# B&R Automation Studio project Template (part 2)

#### slave.fun - functions
```iecst
(********************************************************************
 * COPYRIGHT -- Bernecker + Rainer
 ********************************************************************
 * Program: Slave_00
 * File: Slave_00.fun
 * Author: reischlj
 * Created: March 09, 2011
 ********************************************************************
 * Functions and function blocks of program Slave_00
 ********************************************************************)

FUNCTION Labeler : BOOL
	VAR_INPUT
		Axis : UDINT;
	END_VAR
	VAR_IN_OUT
		AutData : MC_AUTDATA_TYP;
	END_VAR
END_FUNCTION

FUNCTION CrossCutter : BOOL
	VAR_INPUT
		Axis : UDINT;
	END_VAR
	VAR_IN_OUT
		AutData : MC_AUTDATA_TYP;
	END_VAR
END_FUNCTION

FUNCTION FlyingSaw : BOOL
	VAR_INPUT
		Axis  : UDINT;
	END_VAR
	VAR_IN_OUT
		AutData : MC_AUTDATA_TYP;
	END_VAR
END_FUNCTION
```

#### Labeler.st - function
```iecst
(********************************************************************
 * COPYRIGHT -- Bernecker + Rainer
 ********************************************************************
 * PROGRAM: Slave
 * File: Labeler.st
 * Author: Bernecker + Rainer
 * Created: March 01, 2011
 *******************************************************************)

FUNCTION Labeler
    (*general automat parameter*)
        AutData.Master              := Axis;

        AutData.MaxMasterVelocity   := 1000;

    (*Automat STATE 0 Basis State*)

        AutData.State[0].Event[0].Type      := ncST_END;

        AutData.State[0].Event[0].Attribute := ncAT_ONCE;

        AutData.State[0].Event[0].NextState := 1;

    (*Automat STATE 1 Standstill*)

        AutData.State[1].CamProfileIndex    := 16#FFFF;

        AutData.State[1].MasterFactor       := 200;

        AutData.State[1].SlaveFactor        := 0;

        AutData.State[1].CompMode           := ncONLYCOMP;

        AutData.State[1].MasterCompDistance := 800;

        AutData.State[1].SlaveCompDistance  := 0;

        AutData.State[1].Event[0].Type      := ncTRIGGER1+ncP_EDGE;

        AutData.State[1].Event[0].Attribute := ncST_END;

        AutData.State[1].Event[0].NextState := 2;

        AutData.State[1].Event[1].Type      := ncST_END;

        AutData.State[1].Event[1].Attribute := ncST_END;

        AutData.State[1].Event[1].NextState := 1;

    (*Automat STATE 2 Labeling with half compensation*)

        AutData.State[2].CamProfileIndex    := 16#FFFF;

        AutData.State[2].MasterFactor       := 200;

        AutData.State[2].SlaveFactor        := 200;

        AutData.State[2].CompMode           := ncONLYCOMP;
        AutData.State[2].MasterCompDistance := 800;

        AutData.State[2].SlaveCompDistance  := 400;

        AutData.State[2].Event[0].Type      := ncTRIGGER1+ncP_EDGE;

        AutData.State[2].Event[0].Attribute := ncST_END;

        AutData.State[2].Event[0].NextState := 3;

        AutData.State[2].Event[1].Type      := ncST_END;

        AutData.State[2].Event[1].Attribute := ncST_END;

        AutData.State[2].Event[1].NextState := 4;

    (*Automat STATE 3 Labeling *)

        AutData.State[3].CamProfileIndex    := 16#FFFF;

        AutData.State[3].MasterFactor       := 200;

        AutData.State[3].SlaveFactor        := 200;

        AutData.State[3].CompMode           := ncONLYCOMP;

        AutData.State[3].MasterCompDistance := 800;

        AutData.State[3].SlaveCompDistance  := 800;

        AutData.State[3].Event[0].Type      := ncTRIGGER1+ncP_EDGE;

        AutData.State[3].Event[0].Attribute := ncST_END;

        AutData.State[3].Event[0].NextState := 3;

        AutData.State[3].Event[1].Type      := ncST_END;
		AutData.State[3].Event[1].Attribute := ncST_END;
		AutData.State[3].Event[1].NextState := 4;

    (*Automat STATE 4 Return to starting position*)
        AutData.State[4].CamProfileIndex    := 16#FFFF;
        AutData.State[4].MasterFactor       := 200;
        AutData.State[4].SlaveFactor        := 0;
        AutData.State[4].CompMode           := ncONLYCOMP;
        AutData.State[4].MasterCompDistance := 800;
        AutData.State[4].SlaveCompDistance  := 400;

        AutData.State[4].Event[0].Type      := ncTRIGGER1+ncP_EDGE;
        AutData.State[4].Event[0].Attribute := ncST_END;
        AutData.State[4].Event[0].NextState := 2;

        AutData.State[4].Event[1].Type      := ncST_END;
        AutData.State[4].Event[1].Attribute := ncST_END;
        AutData.State[4].Event[1].NextState := 1;

        Labeler := TRUE;
END_FUNCTION
```

#### CrossCutter.st - function
```iecst
(********************************************************************
 * COPYRIGHT -- Bernecker + Rainer
 ********************************************************************
 * PROGRAM: Slave
 * File: CrossCutter.st
 * Author: Bernecker + Rainer
 * Created: March 01, 2011
 *******************************************************************)

FUNCTION CrossCutter
    (*general automat parameter*)
        AutData.Master              := Axis;

        AutData.MaxMasterVelocity   := 1000;

    (*Automat STATE 0 Basis State*)

        AutData.State[0].Event[0].Type      := ncST_END;

        AutData.State[0].Event[0].Attribute := ncAT_ONCE;

        AutData.State[0].Event[0].NextState := 1;

    (*Automat STATE 1 Standstill*)

        AutData.State[1].CamProfileIndex    := 16#FFFE;

        AutData.State[1].MasterFactor       := 200;

        AutData.State[1].SlaveFactor        := 0;
        AutData.State[1].CompMode           := ncWITH_CAM;
        AutData.State[1].MasterCompDistance := 1000;
        AutData.State[1].SlaveCompDistance  := 0;

        AutData.State[1].Event[0].Type      := ncSIGNAL1;
        AutData.State[1].Event[0].Attribute := ncAT_ONCE;
        AutData.State[1].Event[0].NextState := 2;

    (*Automat STATE 2 Move Slave to Cutting Position*)
        AutData.State[2].CamProfileIndex    := 16#FFFF;
        AutData.State[2].MasterFactor       := 200;
        AutData.State[2].SlaveFactor        := 200;
        AutData.State[2].CompMode           := ncWITH_CAM;
        AutData.State[2].MasterCompDistance := 500;
        AutData.State[2].SlaveCompDistance  := 1800;

        AutData.State[2].Event[0].Type      := ncST_END;
        AutData.State[2].Event[0].Attribute := ncST_END;
        AutData.State[2].Event[0].NextState := 3;

    (*Automat STATE 3 Execute one cut every master period*)
        AutData.State[3].CamProfileIndex    := 16#FFFF;
        AutData.State[3].MasterFactor       := 200;
        AutData.State[3].SlaveFactor        := 200;
        AutData.State[3].CompMode           := ncWITH_CAM;
        AutData.State[3].MasterCompDistance := 1000;
        AutData.State[3].SlaveCompDistance  := 3600;

        AutData.State[3].Event[0].Type      := ncSIGNAL2;
        AutData.State[3].Event[0].Attribute := ncST_END;
        AutData.State[3].Event[0].NextState := 4;

        AutData.State[3].Event[1].Type      := ncST_END;
        AutData.State[3].Event[1].Attribute := ncST_END;
        AutData.State[3].Event[1].NextState := 3;

    (*Automat STATE 4 Stop Motion at Starting Point*)
        AutData.State[4].CamProfileIndex    := 16#FFFF;
        AutData.State[4].MasterFactor       := 200;
        AutData.State[4].SlaveFactor        := 0;
        AutData.State[4].CompMode           := ncWITH_CAM;
        AutData.State[4].MasterCompDistance := 500;
        AutData.State[4].SlaveCompDistance  := 1800;

        AutData.State[4].Event[0].Type      := ncST_END;
        AutData.State[4].Event[0].Attribute := ncST_END;
        AutData.State[4].Event[0].NextState := 1;

        CrossCutter := TRUE;
END_FUNCTION
```

#### FlyingSaw.st - function
```iecst
(********************************************************************
 * COPYRIGHT -- Bernecker + Rainer
 ********************************************************************
 * PROGRAM: Slave
 * File: FlyingSaw.st
 * Author: Bernecker + Rainer
 * Created: March 01, 2011
 *******************************************************************)

FUNCTION FlyingSaw
    (*general automat parameters*)
        AutData.Master              := Axis;

        AutData.StartPosition       := 0;

        AutData.StartInterval       := 1000;

        AutData.MaxMasterVelocity   := 1000;

    (*Automat STATE 0 Basis State*)

        AutData.State[0].Event[0].Type      := ncST_END;

        AutData.State[0].Event[0].Attribute := ncAT_ONCE;

        AutData.State[0].Event[0].NextState := 1;

    (*Automat STATE 1 Standstill*)

        AutData.State[1].CamProfileIndex    := 16#FFFF;

        AutData.State[1].MasterFactor       := 200;

        AutData.State[1].SlaveFactor        := 0;

        AutData.State[1].CompMode           := ncONLYCOMP;

        AutData.State[1].MasterCompDistance := 800;

        AutData.State[1].SlaveCompDistance  := 0;

        AutData.State[1].Event[0].Type      := ncS_START;

        AutData.State[1].Event[0].Attribute := ncAT_ONCE;

        AutData.State[1].Event[0].NextState := 2;

    (*Autoamt STATE 2 Synchronous movement*)
        AutData.State[2].CamProfileIndex    := 16#FFFF;
        AutData.State[2].MasterFactor       := 500;
        AutData.State[2].SlaveFactor        := 500;
        AutData.State[2].CompMode           := ncONLYCOMP;
        AutData.State[2].MasterCompDistance := 100;
        AutData.State[2].SlaveCompDistance  := 100;

        AutData.State[2].Event[0].Type      := ncST_END;
        AutData.State[2].Event[0].Attribute := ncST_END;
        AutData.State[2].Event[0].NextState := 3;

    (*Automat STATE 3 Return to starting position*)
        AutData.State[3].CamProfileIndex    := 16#FFFF;
        AutData.State[3].MasterFactor       := 100;
        AutData.State[3].SlaveFactor        := 0;
        AutData.State[3].CompMode           := ncONLYCOMP;
        AutData.State[3].MasterCompDistance := 800;
        AutData.State[3].SlaveCompDistance  := -600;

        AutData.State[3].Event[0].Type      := ncST_END;
        AutData.State[3].Event[0].Attribute := ncST_END;
        AutData.State[3].Event[0].NextState := 1;

        FlyingSaw := TRUE;
END_FUNCTION
```

### Program Logical/LibACP10MC_MotionControl_ST/ErrorHandling (IEC) - error handling task

#### errorHandlingCyclic.st - Cyclic code
```iecst
(********************************************************************
 * COPYRIGHT -- Bernecker + Rainer
 ********************************************************************
 * Program: ErrorHandling
 * File: errorHandlingCyclic.st
 * Author: Bernecker + Rainer
 * Created: March 01, 2011
 ********************************************************************
 * Implementation of program Errorhandling
 ********************************************************************)

PROGRAM _CYCLIC

(******************************ERROR_CHECK***************************)
(* check if one of the used FBs reports an error *)
IF ((MC_BR_AxisErrorCollector_0.Error = TRUE) OR (MC_Reset_0.Error = TRUE)) THEN
    ErrorStep := STATE_INTERNAL_ERROR;
END_IF

FOR configAxisIndex := 0 TO TOTAL_AXES BY 1 DO
    IF ((MC_BR_ReadAxisError_0[configAxisIndex].Error = TRUE) OR (MC_ReadStatus_0[configAxisIndex].Error = TRUE)) THEN
        ErrorStep := STATE_INTERNAL_ERROR;
        EXIT;
    END_IF
END_FOR

CASE ErrorStep OF

(**************************** CONFIGURATE_FBS ***********************)
    STATE_CONFIG_FBS: (* configurate the used FBs for the error handling *)
        MC_BR_AxisErrorCollector_0.Axis := mcALL_AXES;
        MC_BR_AxisErrorCollector_0.Enable := TRUE;

        (* configuration the MC_BR_ReadAxisError_0-FBs for all single axes *)
        FOR axisIndex := 0 TO (AXIS_MAX_INDEX) BY 1 DO
            MC_BR_ReadAxisError_0[axisIndex].Axis := AxisRef[axisIndex];
            MC_BR_ReadAxisError_0[axisIndex].Enable := TRUE;
            MC_BR_ReadAxisError_0[axisIndex].Configuration.Format := mcWRAP;
            MC_BR_ReadAxisError_0[axisIndex].Configuration.LineLength := SIZEOF(Axis[axisIndex].Error.ErrorText[0]);
            MC_BR_ReadAxisError_0[axisIndex].Configuration.DataLength := SIZEOF(Axis[axisIndex].Error.ErrorText);
            MC_BR_ReadAxisError_0[axisIndex].Configuration.DataAddress := ADR(Axis[axisIndex].Error.ErrorText[0]);
            MC_BR_ReadAxisError_0[axisIndex].Configuration.DataObjectName :='acp10etxen';
            MC_BR_ReadAxisError_0[axisIndex].Mode := mcTEXT;

            MC_ReadStatus_0[axisIndex].Axis := AxisRef[axisIndex];
            MC_ReadStatus_0[axisIndex].Enable := TRUE;
        END_FOR

        (* configuration the MC_BR_ReadAxisError_0-FBs for all master axes *)
        FOR masterIndex := 0 TO (MASTER_MAX_INDEX) BY 1 DO
            MC_BR_ReadAxisError_0[masterIndex+AXIS_NUMBER].Axis := MasterRef[masterIndex];
            MC_BR_ReadAxisError_0[masterIndex+AXIS_NUMBER].Enable := TRUE;
            MC_BR_ReadAxisError_0[masterIndex+AXIS_NUMBER].Configuration.Format := mcWRAP;
            MC_BR_ReadAxisError_0[masterIndex+AXIS_NUMBER].Configuration.LineLength := SIZEOF(Master[masterIndex].Error.ErrorText[0]);
            MC_BR_ReadAxisError_0[masterIndex+AXIS_NUMBER].Configuration.DataLength := SIZEOF(Master[masterIndex].Error.ErrorText);
            MC_BR_ReadAxisError_0[masterIndex+AXIS_NUMBER].Configuration.DataAddress := ADR(Master[masterIndex].Error.ErrorText[0]);
            MC_BR_ReadAxisError_0[masterIndex+AXIS_NUMBER].Configuration.DataObjectName := 'acp10etxen';
            MC_BR_ReadAxisError_0[masterIndex+AXIS_NUMBER].Mode := mcTEXT;

            MC_ReadStatus_0[masterIndex+AXIS_NUMBER].Axis := MasterRef[masterIndex];
            MC_ReadStatus_0[masterIndex+AXIS_NUMBER].Enable := TRUE;
        END_FOR

        (* configuration the MC_BR_ReadAxisError_0-FBs for all slave axes *)
        FOR slaveIndex := 0 TO (SLAVE_MAX_INDEX) BY 1 DO
            MC_BR_ReadAxisError_0[slaveIndex+AXIS_NUMBER+MASTER_NUMBER].Axis := SlaveRef[slaveIndex];
            MC_BR_ReadAxisError_0[slaveIndex+AXIS_NUMBER+MASTER_NUMBER].Enable := TRUE;
            MC_BR_ReadAxisError_0[slaveIndex+AXIS_NUMBER+MASTER_NUMBER].Configuration.Format := mcWRAP;
            MC_BR_ReadAxisError_0[slaveIndex+AXIS_NUMBER+MASTER_NUMBER].Configuration.LineLength := SIZEOF(Slave[slaveIndex].Error.ErrorText[0]);
            MC_BR_ReadAxisError_0[slaveIndex+AXIS_NUMBER+MASTER_NUMBER].Configuration.DataLength := SIZEOF(Slave[slaveIndex].Error.ErrorText);
            MC_BR_ReadAxisError_0[slaveIndex+AXIS_NUMBER+MASTER_NUMBER].Configuration.DataAddress := ADR(Slave[slaveIndex].Error.ErrorText[0]);
            MC_BR_ReadAxisError_0[slaveIndex+AXIS_NUMBER+MASTER_NUMBER].Configuration.DataObjectName := 'acp10etxen';
            MC_BR_ReadAxisError_0[slaveIndex+AXIS_NUMBER+MASTER_NUMBER].Mode := mcTEXT;

            MC_ReadStatus_0[slaveIndex+AXIS_NUMBER+MASTER_NUMBER].Axis := SlaveRef[slaveIndex];
            MC_ReadStatus_0[slaveIndex+AXIS_NUMBER+MASTER_NUMBER].Enable := TRUE;
        END_FOR

        (* configuration the MC_BR_ReadAxisError_0-FBs for all power supply module *)
        FOR psmIndex := 0 TO (PSM_MAX_INDEX) BY 1 DO
            MC_BR_ReadAxisError_0[psmIndex+AXIS_NUMBER+MASTER_NUMBER+SLAVE_NUMBER].Axis := PsmRef[psmIndex];
            MC_BR_ReadAxisError_0[psmIndex+AXIS_NUMBER+MASTER_NUMBER+SLAVE_NUMBER].Enable := TRUE;
            MC_BR_ReadAxisError_0[psmIndex+AXIS_NUMBER+MASTER_NUMBER+SLAVE_NUMBER].Configuration.Format := mcWRAP;
            MC_BR_ReadAxisError_0[psmIndex+AXIS_NUMBER+MASTER_NUMBER+SLAVE_NUMBER].Configuration.LineLength := SIZEOF(PowerSupply[psmIndex].Error.ErrorText[0]);
            MC_BR_ReadAxisError_0[psmIndex+AXIS_NUMBER+MASTER_NUMBER+SLAVE_NUMBER].Configuration.DataLength := SIZEOF(PowerSupply[psmIndex].Error.ErrorText);
            MC_BR_ReadAxisError_0[psmIndex+AXIS_NUMBER+MASTER_NUMBER+SLAVE_NUMBER].Configuration.DataAddress := ADR(PowerSupply[psmIndex].Error.ErrorText[0]);
            MC_BR_ReadAxisError_0[psmIndex+AXIS_NUMBER+MASTER_NUMBER+SLAVE_NUMBER].Configuration.DataObjectName := 'acp10etxen';
            MC_BR_ReadAxisError_0[psmIndex+AXIS_NUMBER+MASTER_NUMBER+SLAVE_NUMBER].Mode := mcTEXT;

            MC_ReadStatus_0[psmIndex+AXIS_NUMBER+MASTER_NUMBER+SLAVE_NUMBER].Axis := PsmRef[psmIndex];
            MC_ReadStatus_0[psmIndex+AXIS_NUMBER+MASTER_NUMBER+SLAVE_NUMBER].Enable := TRUE;
        END_FOR

        ErrorStep := STATE_WAIT;
        AcknowledgeStep := STATE_ERROR_SCAN;

        (* End of STATE_CONFIG_FBS *)

(*************************** CHECK_AXES_FOR_ERROR *******************)
    STATE_WAIT: (* check if at least on one of the axes an error occured *)
        IF ((MC_BR_AxisErrorCollector_0.AxisError = TRUE) OR
            (MC_BR_AxisErrorCollector_0.AxisWarning = TRUE) OR
            (MC_BR_AxisErrorCollector_0.FunctionBlockError = TRUE) OR
            (MC_BR_AxisErrorCollector_0.Errorstop = TRUE)) THEN
              ErrorStep := STATE_ERROR_HANDLING;
        ELSE
            GlobalError.AxisTyp := '';
            GlobalError.AxisIndex := 0;
            GlobalError.ErrorRecord.Info := 0;
            GlobalError.ErrorRecord.Number := 0;
            GlobalError.ErrorRecord.ParID := 0;
            GlobalError.ErrorText[0] := '';
            GlobalError.ErrorText[1] := '';
            GlobalError.ErrorText[2] := '';
            GlobalError.ErrorText[3] := '';
        END_IF

        (* End of STATE_WAIT *)

(**************************** HANDLE_ACTIVE_ERRORS ******************)
    STATE_ERROR_HANDLING: (* check witch axis is in ErrorStop and withc axes has to be stopped *)
        (* check if a single axis has to be stopped *)
        FOR axisIndex := 0 TO (AXIS_MAX_INDEX) BY 1 DO
            IF (MC_ReadStatus_0[axisIndex].Errorstop = TRUE) THEN
                Axis[axisIndex].Command.Stop := TRUE;
            END_IF
        END_FOR

        (* check if the master slave combination has to be stopped *)
        FOR masterIndex := 0 TO (MASTER_MAX_INDEX) BY 1 DO
            IF (MC_ReadStatus_0[masterIndex+AXIS_NUMBER].Errorstop = TRUE) THEN
                FOR masterIndex := 0 TO (MASTER_MAX_INDEX) BY 1 DO
                    Master[masterIndex].Command.Stop := TRUE;
                END_FOR

                FOR slaveIndex := 0 TO (SLAVE_MAX_INDEX) BY 1 DO
                    Slave[slaveIndex].Command.Stop := TRUE;
                END_FOR
            END_IF
        END_FOR

        (* check if the master slave combination has to be stopped *)
        FOR slaveIndex := 0 TO (SLAVE_MAX_INDEX) BY 1 DO
            IF  (MC_ReadStatus_0[slaveIndex+AXIS_NUMBER+MASTER_NUMBER].Errorstop = TRUE) THEN
                FOR masterIndex := 0 TO (MASTER_MAX_INDEX) BY 1 DO
                    Master[masterIndex].Command.Stop := TRUE;
                END_FOR

                FOR slaveIndex := 0 TO (SLAVE_MAX_INDEX) BY 1 DO
                    Slave[slaveIndex].Command.Stop := TRUE;
                END_FOR
            END_IF
        END_FOR

    (******************* STEP_SEQUENCE OF ERROR ACKNOWLEDGE *************)
    CASE AcknowledgeStep OF
        (************************** SEARCH FOR ERRORS ***********************)
        STATE_ERROR_SCAN: (* check if an error is active on one of the axis *)
            ErrorStep := STATE_WAIT;
            FOR totalAxisIndex := 0 TO (TOTAL_AXES-1) BY 1 DO
                IF ((MC_BR_ReadAxisError_0[totalAxisIndex].AxisErrorCount > 0) OR
                    (MC_BR_ReadAxisError_0[totalAxisIndex].AxisWarningCount > 0) OR
                    (MC_BR_ReadAxisError_0[totalAxisIndex].FunctionBlockErrorCount > 0)) THEN
                    AcknowledgeStep := STATE_ERROR_ACKNOWLEDGE;
                    ErrorStep := STATE_ERROR_HANDLING;
                    EXIT;
                ELSIF (MC_ReadStatus_0[totalAxisIndex].Errorstop = TRUE) THEN
                    AcknowledgeStep := STATE_RESET;
                    ErrorStep := STATE_ERROR_HANDLING;
                    EXIT;
                END_IF
            END_FOR

            (* End of STATE_ERROR_SCAN *)

        (********************** WAIT FOR ACKNOWLEDGE ************************)
        STATE_ERROR_ACKNOWLEDGE:
            (* copy the actual error information to the global error structure *)
            IF (totalAxisIndex < AXIS_NUMBER) THEN
                GlobalError.AxisTyp := 'Axis';
                GlobalError.ErrorText := Axis[totalAxisIndex].Error.ErrorText;
                GlobalError.ErrorRecord := Axis[totalAxisIndex].Error.ErrorRecord;
            ELSIF (totalAxisIndex < (AXIS_NUMBER+MASTER_NUMBER)) THEN
                GlobalError.AxisTyp := 'Master';
                GlobalError.ErrorText := Master[totalAxisIndex-AXIS_NUMBER].Error.ErrorText;
                GlobalError.ErrorRecord := Master[totalAxisIndex-AXIS_NUMBER].Error.ErrorRecord;
            ELSIF (totalAxisIndex < (AXIS_NUMBER+MASTER_NUMBER+SLAVE_NUMBER)) THEN
                GlobalError.AxisTyp := 'Slave';
                GlobalError.ErrorText := Slave[totalAxisIndex-(AXIS_NUMBER+MASTER_NUMBER)].Error.ErrorText;
                GlobalError.ErrorRecord := Slave[totalAxisIndex-(AXIS_NUMBER+MASTER_NUMBER)].Error.ErrorRecord;
            ELSIF (totalAxisIndex < (AXIS_NUMBER+MASTER_NUMBER+SLAVE_NUMBER+PSM_NUMBER)) THEN
                GlobalError.AxisTyp := 'PSM';
                GlobalError.ErrorText := PowerSupply[totalAxisIndex-(AXIS_NUMBER+MASTER_NUMBER+SLAVE_NUMBER)].Error.ErrorText;
                GlobalError.ErrorRecord := PowerSupply[totalAxisIndex-(AXIS_NUMBER+MASTER_NUMBER+SLAVE_NUMBER)].Error.ErrorRecord;
            END_IF
            GlobalError.AxisIndex := totalAxisIndex;

            IF (GlobalCommand.ErrorAcknowledge = TRUE) THEN
                GlobalCommand.ErrorAcknowledge := FALSE;
                MC_BR_ReadAxisError_0[totalAxisIndex].Acknowledge := TRUE;
            ELSIF (MC_BR_ReadAxisError_0[totalAxisIndex].Acknowledge = TRUE) THEN
                MC_BR_ReadAxisError_0[totalAxisIndex].Acknowledge := FALSE;
                AcknowledgeStep := STATE_ERROR_SCAN;
            END_IF

            (* End of STATE_ERROR_ACKNOWLEDGE *)

        (************************* RESET AXES IN ERRORSTEP ******************)
        STATE_RESET:
            IF (totalAxisIndex < AXIS_NUMBER) THEN
                MC_Reset_0.Axis := AxisRef[totalAxisIndex];
            ELSIF (totalAxisIndex < (AXIS_NUMBER+MASTER_NUMBER)) THEN
                MC_Reset_0.Axis := MasterRef[totalAxisIndex-AXIS_NUMBER];
            ELSIF (totalAxisIndex < (AXIS_NUMBER+MASTER_NUMBER+SLAVE_NUMBER)) THEN
                MC_Reset_0.Axis := SlaveRef[totalAxisIndex-(AXIS_NUMBER+MASTER_NUMBER)];
            ELSE
                MC_Reset_0.Axis := PsmRef[totalAxisIndex-(AXIS_NUMBER+MASTER_NUMBER+SLAVE_NUMBER)];
            END_IF
            MC_Reset_0.Execute := TRUE;

            IF (MC_Reset_0.Done = TRUE) THEN
                MC_Reset_0.Execute := 0;
                AcknowledgeStep := STATE_ERROR_SCAN;
            END_IF

            (* End of STATE_RESET *)
    END_CASE
    (************* END OF STEP SEQUENCE OF ERROR ACKNOWLEDGE ************)

    (* End of STATE_ERROR_HANDLING *)

(****************** DEACTIVATE USED FBS IN CASE OF ERROR ************)
    STATE_INTERNAL_ERROR:
        MC_BR_AxisErrorCollector_0.Enable := FALSE;
        MC_Reset_0.Execute := FALSE;

        FOR configAxisIndex := 0 TO (TOTAL_AXES-1) BY 1 DO
            MC_BR_ReadAxisError_0[configAxisIndex].Enable := FALSE;
            MC_ReadStatus_0[configAxisIndex].Enable := FALSE;
        END_FOR

        ErrorStep := STATE_CONFIG_FBS;

        (* End of STATE_INTERNAL_ERROR *)

END_CASE

(************************** CALL FBS ********************************)
MC_BR_AxisErrorCollector_0();

FOR configAxisIndex := 0 TO TOTAL_AXES BY 1 DO
    MC_BR_ReadAxisError_0[configAxisIndex]();
    IF (configAxisIndex < AXIS_NUMBER) THEN
        Axis[configAxisIndex].Error.AxisErrorCount := MC_BR_ReadAxisError_0[configAxisIndex].AxisErrorCount;
        Axis[configAxisIndex].Error.AxisWarningCount := MC_BR_ReadAxisError_0[configAxisIndex].AxisWarningCount;
        Axis[configAxisIndex].Error.FunctionBlockErrorCount := MC_BR_ReadAxisError_0[configAxisIndex].FunctionBlockErrorCount;
        Axis[configAxisIndex].Error.ErrorRecord := MC_BR_ReadAxisError_0[configAxisIndex].ErrorRecord;
    ELSIF (configAxisIndex < (AXIS_NUMBER+MASTER_NUMBER)) THEN
        Master[configAxisIndex-AXIS_NUMBER].Error.AxisErrorCount := MC_BR_ReadAxisError_0[configAxisIndex].AxisErrorCount;
        Master[configAxisIndex-AXIS_NUMBER].Error.AxisWarningCount := MC_BR_ReadAxisError_0[configAxisIndex].AxisWarningCount;
        Master[configAxisIndex-AXIS_NUMBER].Error.FunctionBlockErrorCount := MC_BR_ReadAxisError_0[configAxisIndex].FunctionBlockErrorCount;
        Master[configAxisIndex-AXIS_NUMBER].Error.ErrorRecord := MC_BR_ReadAxisError_0[configAxisIndex].ErrorRecord;
	ELSIF (configAxisIndex < (AXIS_NUMBER+MASTER_NUMBER+SLAVE_NUMBER)) THEN
		Slave[configAxisIndex-(AXIS_NUMBER+MASTER_NUMBER)].Error.AxisErrorCount := MC_BR_ReadAxisError_0[configAxisIndex].AxisErrorCount;
		Slave[configAxisIndex-(AXIS_NUMBER+MASTER_NUMBER)].Error.AxisWarningCount := MC_BR_ReadAxisError_0[configAxisIndex].AxisWarningCount;
		Slave[configAxisIndex-(AXIS_NUMBER+MASTER_NUMBER)].Error.FunctionBlockErrorCount := MC_BR_ReadAxisError_0[configAxisIndex].FunctionBlockErrorCount;
		Slave[configAxisIndex-(AXIS_NUMBER+MASTER_NUMBER)].Error.ErrorRecord := MC_BR_ReadAxisError_0[configAxisIndex].ErrorRecord;
	ELSIF (configAxisIndex < (AXIS_NUMBER+MASTER_NUMBER+SLAVE_NUMBER+PSM_NUMBER)) THEN
		PowerSupply[configAxisIndex-(AXIS_NUMBER+MASTER_NUMBER+SLAVE_NUMBER)].Error.AxisErrorCount := MC_BR_ReadAxisError_0[configAxisIndex].AxisErrorCount;
        PowerSupply[configAxisIndex-(AXIS_NUMBER+MASTER_NUMBER+SLAVE_NUMBER)].Error.AxisWarningCount := MC_BR_ReadAxisError_0[configAxisIndex].AxisWarningCount;
        PowerSupply[configAxisIndex-(AXIS_NUMBER+MASTER_NUMBER+SLAVE_NUMBER)].Error.FunctionBlockErrorCount := MC_BR_ReadAxisError_0[configAxisIndex].FunctionBlockErrorCount;
        PowerSupply[configAxisIndex-(AXIS_NUMBER+MASTER_NUMBER+SLAVE_NUMBER)].Error.ErrorRecord := MC_BR_ReadAxisError_0[configAxisIndex].ErrorRecord;
    END_IF
    MC_ReadStatus_0[configAxisIndex]();
END_FOR

MC_Reset_0();

END_PROGRAM
```

#### errorHandlingInit.st - Initialization code
```iecst
(********************************************************************
 * COPYRIGHT -- Bernecker + Rainer
 ********************************************************************
 * Program: ErrorHandling
 * File: errorHandlingInit.st
 * Author: Bernecker + Rainer
 * Created: March 01, 2011
 ********************************************************************
  * Implementation OF PROGRAM ErrorHandling
 ********************************************************************)

PROGRAM _INIT
    AcknowledgeStep := STATE_ERROR_SCAN;
END_PROGRAM
```

#### errorHandling.var - Local variables
```iecst
(*Index variables*)
VAR
	configAxisIndex : USINT; (*count variable for configurating "for"-loops*)
	totalAxisIndex : USINT; (*count variable for all axes acting "for"-loops*)
	psmIndex : USINT;
	axisIndex : USINT; (*count variable for single axes acting "for"-loops*)
	masterIndex : USINT; (*count variable for master axes acting "for"-loops*)
	slaveIndex : USINT; (*count variable for slave axes acting "for"-loops*)
END_VAR
(*Actual steps inside the step sequences*)
VAR
	ErrorStep : USINT; (*current step in the step sequence*)
	AcknowledgeStep : USINT; (*current step in the acknowledge step sequence *)
END_VAR
(*Error Steps*)
VAR CONSTANT
	STATE_CONFIG_FBS : USINT := 0; (*constant for the step in which the function blocks are configured*)
	STATE_WAIT : USINT := 1; (*constant for the step in which it is waited for a occuring error*)
	STATE_ERROR_HANDLING : USINT := 2; (*constant for the step in which all necessary axes are stopped *)
	STATE_INTERNAL_ERROR : USINT := 3; (*constant for the step in which all function blocks are disabled in case of an FB error*)
END_VAR
(*Acknowledge Steps*)
VAR CONSTANT
	STATE_ERROR_SCAN : USINT := 10; (*constant for the step in which the first active is searched*)
	STATE_ERROR_ACKNOWLEDGE : USINT := 11; (*constant for the step in which the actual output error is acknowledged after user command*)
	STATE_RESET : USINT := 12; (*constant for the step in which the axes are reset after all errors where acknowled*)
END_VAR
(*Function Blocks*)
VAR
	MC_BR_AxisErrorCollector_0 : MC_BR_AxisErrorCollector; (*Function Block*)
	MC_BR_ReadAxisError_0 : ARRAY[0..TOTAL_AXES] OF MC_BR_ReadAxisError; (*Function Block*)
	MC_ReadStatus_0 : ARRAY[0..TOTAL_AXES] OF MC_ReadStatus; (*Function Block*)
	MC_Reset_0 : MC_Reset; (*Function Block*)
END_VAR
```
